TYPE SQL_Get_Payload_Struct :
STRUCT
	// 
	Payload_Uid : STRING(36);
	PosBegain	: LREAL;
	PosEnd	: LREAL;
END_STRUCT
END_TYPE

(* stored: Version 1.1.0.1, ProductVersion 3.1.4026.13
   DUT SQL_Get_Payload_Struct: Id {656b129a-eaea-4fc3-ae2d-e814525d2b51} *)
